RoboDK station: Stringer A-BotDOWN-BOX1.rdk

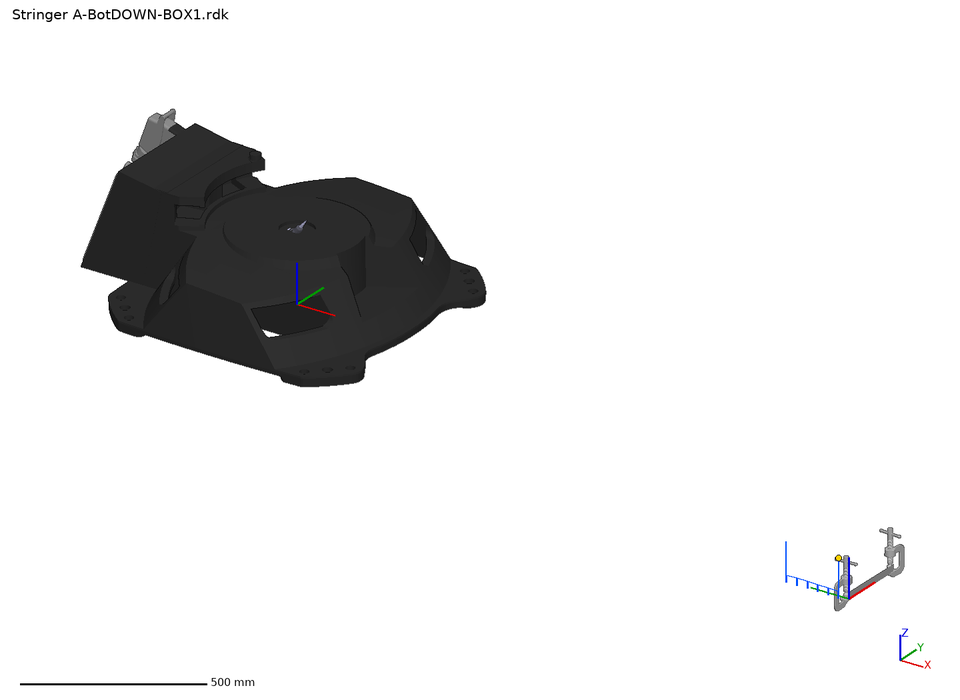
[picture v0: the station drawn from its stored meshes, robots at their saved joint values, targets as dots, program paths as lines]
Station Stringer A-BotDOWN-BOX1 (saved by RoboDK 5.2.3). Poses are relative to the parent item; angles as X-Y-Z fixed-axis rotations.
  - frame KUKA KR 210 R2700 extra Base at (0, 0, 0) mm
    - robot KUKA KR 210 R2700 extra: 6 axes, payload 210 kg, reach 2696 mm, repeatability 0.06 mm, weight 1068 kg
        joint limits [-185, -140, -120, -350, -125, -350] to [185, -5, 155, 350, 125, 350]; home [0, -90, 90, 0, 0, 0]; saved at [-7.358, -33.904, 111.259, 169.595, 26.502, -176.398]
      - tool Spindle, TCP at (32, 0, 260) mm, rotated rx 0 ry 39 rz 0 deg, size 157.3 x 72 x 259.9 mm
  - frame Frame 2 at (1800, 0, -372.68) mm, rotated rx 0 ry 0 rz 90 deg
    - object L-Stringer A - bot down at (0, 0, 0) mm, size 219.8 x 20 x 20 mm, geometry from L-Stringer A - bot down.stl
    - object Stringer A-BotDOWN-BOX1 at (0, 0, 0) mm, rotated rx 0 ry 0 rz -90 deg, 6 curves, geometry from Point 6
  - machining project Point settings: rotZ(0) | rotX(0)*rotY(0) | rotz(0) | onStart | onPathStart | onApproach | onPoint | onRetract | onFinish | SetRPM(%1) | SetTool(%1) | Extruder(%1) | default | default | OutOnMov(%1) | OutOffMov(%1) | onPathFinish | M_RunCode(%1) | riverData=C:\Windows\System32\Driv | PS_BROWSER_APP_PROFILE_STRING=Inter | PS_BROWSER_USER_PROFILE_STRING=Defa | OCALAPPDATA=C:\Users\jbert\AppData\Loc | OneDrive=C:\Users\jbert\O | Path=C:\Program Files (x86)\NVIDIA Corpora
  - program Point (41 instructions, listed below)
  - object FinalClamp at (1787.61, 4.47, -310.38) mm, rotated rx 163.76 ry 89.17 rz -12.8 deg, size 145.3 x 71.1 x 72 mm, geometry from FinalClamp.stp
  - object FinalClamp2 at (1783.24, 215.04, -312.43) mm, rotated rx -65.04 ry 88.51 rz -68.16 deg, size 145.3 x 71.1 x 72 mm, geometry from FinalClamp.stp
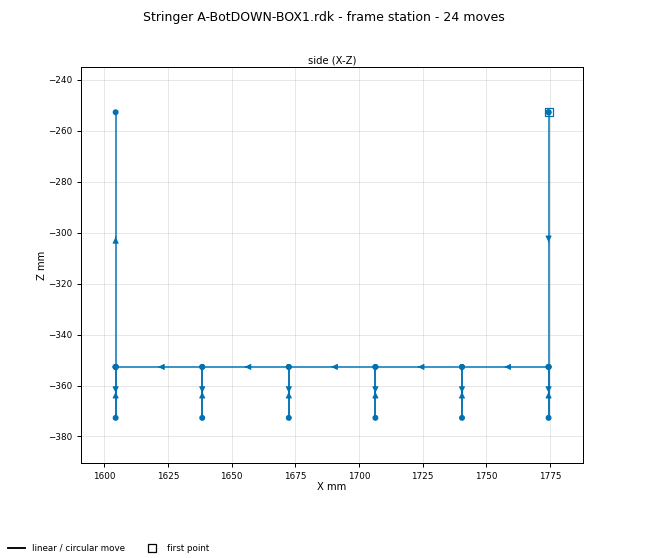
[picture p0: tool path of Stringer A-BotDOWN-BOX1.rdk in frame station, 24 of 24 moves have a stored position in this frame; points joined in program order, loops and branches not executed]

--- program Point (robot KUKA KR 210 R2700 extra) ---
  Smooth(1)
  Set speed (1000.0 mm/s)
  Set Ref.: Frame 2
  Set Tool: Spindle
  Show Spindle
  MoveJ 1 to (-11.37, 25.57, 120) mm, rotated rx -180 ry 0 rz -180 deg; joints [-0.967, -34.025, 111.914, 178.654, 26.891, -179.551]
  MoveL 2 to (-11.37, 25.57, 120) mm, rotated rx -180 ry 0 rz -180 deg; joints [-0.967, -34.025, 111.914, 178.654, 26.891, -179.551]
  MoveL 3 to (-11.37, 25.57, 20) mm, rotated rx 180 ry 0 rz 180 deg; joints [-0.967, -28.692, 109.271, 178.767, 29.58, -179.679]
  MoveL 4 to (-11.37, 25.57, 20) mm, rotated rx 180 ry 0 rz 180 deg; joints [-0.967, -28.692, 109.271, 178.767, 29.58, -179.679]
  Set speed (50.0 mm/s)
  MoveL 5 to (-11.37, 25.57, 0) mm, rotated rx -180 ry 0 rz -180 deg; joints [-0.967, -27.634, 108.694, 178.785, 30.062, -179.7]
  MoveL 6 to (-11.37, 25.57, 20) mm, rotated rx 180 ry 0 rz 180 deg; joints [-0.967, -28.692, 109.271, 178.767, 29.58, -179.679]
  Set speed (1000.0 mm/s)
  MoveL 7 to (-11.37, 59.57, 20) mm, rotated rx -180 ry 0 rz -180 deg; joints [-2.252, -28.686, 109.221, 177.125, 29.545, -179.249]
  Set speed (50.0 mm/s)
  MoveL 8 to (-11.37, 59.57, 0) mm, rotated rx -180 ry 0 rz -180 deg; joints [-2.252, -27.628, 108.645, 177.167, 30.026, -179.297]
  MoveL 9 to (-11.37, 59.57, 20) mm, rotated rx -180 ry 0 rz -180 deg; joints [-2.252, -28.686, 109.221, 177.125, 29.545, -179.249]
  Set speed (1000.0 mm/s)
  MoveL 10 to (-11.37, 93.57, 20) mm, rotated rx 180 ry 0 rz -180 deg; joints [-3.535, -28.674, 109.132, 175.478, 29.481, -178.81]
  Set speed (50.0 mm/s)
  MoveL 11 to (-11.37, 93.57, 0) mm, rotated rx -180 ry 0 rz -180 deg; joints [-3.535, -27.617, 108.556, 175.544, 29.961, -178.886]
  MoveL 12 to (-11.37, 93.57, 20) mm, rotated rx 180 ry 0 rz -180 deg; joints [-3.535, -28.674, 109.132, 175.478, 29.481, -178.81]
  Set speed (1000.0 mm/s)
  MoveL 13 to (-11.37, 127.57, 20) mm, rotated rx 180 ry 0 rz 180 deg; joints [-4.815, -28.656, 109.003, 173.821, 29.391, -178.357]
  Set speed (50.0 mm/s)
  MoveL 14 to (-11.37, 127.57, 0) mm, rotated rx 180 ry 0 rz -180 deg; joints [-4.815, -27.6, 108.428, 173.912, 29.869, -178.461]
  MoveL 15 to (-11.37, 127.57, 20) mm, rotated rx 180 ry 0 rz 180 deg; joints [-4.815, -28.656, 109.003, 173.821, 29.391, -178.357]
  Set speed (1000.0 mm/s)
  MoveL 16 to (-11.37, 161.57, 20) mm, rotated rx -180 ry 0 rz -180 deg; joints [-6.089, -28.633, 108.835, 172.153, 29.273, -177.884]
  Set speed (50.0 mm/s)
  MoveL 17 to (-11.37, 161.57, 0) mm, rotated rx 180 ry 0 rz -180 deg; joints [-6.089, -27.578, 108.261, 172.268, 29.749, -178.016]
  MoveL 18 to (-11.37, 161.57, 20) mm, rotated rx -180 ry 0 rz -180 deg; joints [-6.089, -28.633, 108.835, 172.153, 29.273, -177.884]
  Set speed (1000.0 mm/s)
  MoveL 19 to (-11.37, 195.57, 20) mm, rotated rx 180 ry 0 rz 180 deg; joints [-7.358, -28.604, 108.628, 170.47, 29.13, -177.388]
  Set speed (50.0 mm/s)
  MoveL 20 to (-11.37, 195.57, 0) mm, rotated rx 180 ry 0 rz 180 deg; joints [-7.358, -27.551, 108.054, 170.61, 29.602, -177.548]
  MoveL 21 to (-11.37, 195.57, 20) mm, rotated rx 180 ry 0 rz 180 deg; joints [-7.358, -28.604, 108.628, 170.47, 29.13, -177.388]
  MoveL 22 to (-11.37, 195.57, 20) mm, rotated rx 180 ry 0 rz 180 deg; joints [-7.358, -28.604, 108.628, 170.47, 29.13, -177.388]
  Set speed (1000.0 mm/s)
  MoveL 23 to (-11.37, 195.57, 20) mm, rotated rx 180 ry 0 rz 180 deg; joints [-7.358, -28.604, 108.628, 170.47, 29.13, -177.388]
  MoveL 24 to (-11.37, 195.57, 120) mm, rotated rx 180 ry 0 rz 180 deg; joints [-7.358, -33.904, 111.259, 169.595, 26.502, -176.398]
